// Mitsubishi GX Works2 project: sftEx01   PLC: Q02/Q02H

PROGRAM MAIN
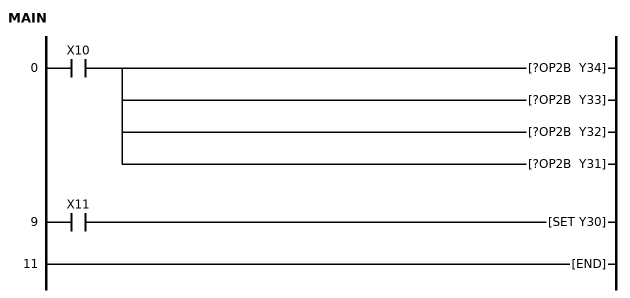
0     LD      X10
      ?OP2B   Y34
      ?OP2B   Y33
      ?OP2B   Y32
      ?OP2B   Y31
9     LD      X11
      SET     Y30
11    END
END_PROGRAM
